// TwinCAT 3 PLC project StopLight
// ProgramVersion: 3.1.4024.0
// libraries:
//   Tc2_Standard, * (Beckhoff Automation GmbH)
//   Tc2_System, * (Beckhoff Automation GmbH)
//   Tc3_Module, * (Beckhoff Automation GmbH)
// project tree:
//   / PlcTask.TcTTO
//   POUs/ MAIN.TcPOU
// real-time tasks:
//   TASK PlcTask: cycle T#10ms, priority 20, ADS port 350

CONFIGURATION StopLight
    RESOURCE PLC ON TwinCAT3
        TASK PlcTask(INTERVAL := T#10ms, PRIORITY := 20);
        PROGRAM MAIN WITH PlcTask : MAIN;
    END_RESOURCE
END_CONFIGURATION

// ---- POUs/MAIN.TcPOU
PROGRAM MAIN
VAR
	gGreenlight : BOOL := FALSE;
	yYellowlight : BOOL := FALSE;
	rRedLight : BOOL := FALSE;
	gGreenlighttimer : TON;
	yYellowlighttimer : TON;
	rRedlighttimer : TON;
END_VAR

gGreenlighttimer(IN := NOT rRedlighttimer.Q, PT := T#5S);

yYellowlighttimer(IN := gGreenlighttimer.Q, PT := T#2S);

rRedlighttimer(IN := yYellowlighttimer.Q, PT := T#5S);

gGreenlight := NOT gGreenlighttimer.Q AND gGreenlighttimer.IN;

yYellowlight := NOT yYellowlighttimer.Q AND yYellowlighttimer.IN;

rRedLight := NOT rRedlighttimer.Q AND rRedlighttimer.IN;

END_PROGRAM
